FUNCTION_BLOCK FB_BaseHMILoggerElement_Command
VAR
	stDataCheck					: ST_BaseHMILoggerElement_Command_DataCheck;

END_VAR

END_FUNCTION_BLOCK

(* stored: Version 1.1.0.1
   POU FB_BaseHMILoggerElement_Command: Id {8f426e87-d199-0feb-30a3-798673a26f74}, SpecialFunc None *)
